// Mitsubishi GX Works2 project: fx1nc_test_in_out   PLC: FX1N/FX1NC

PROGRAM MAIN
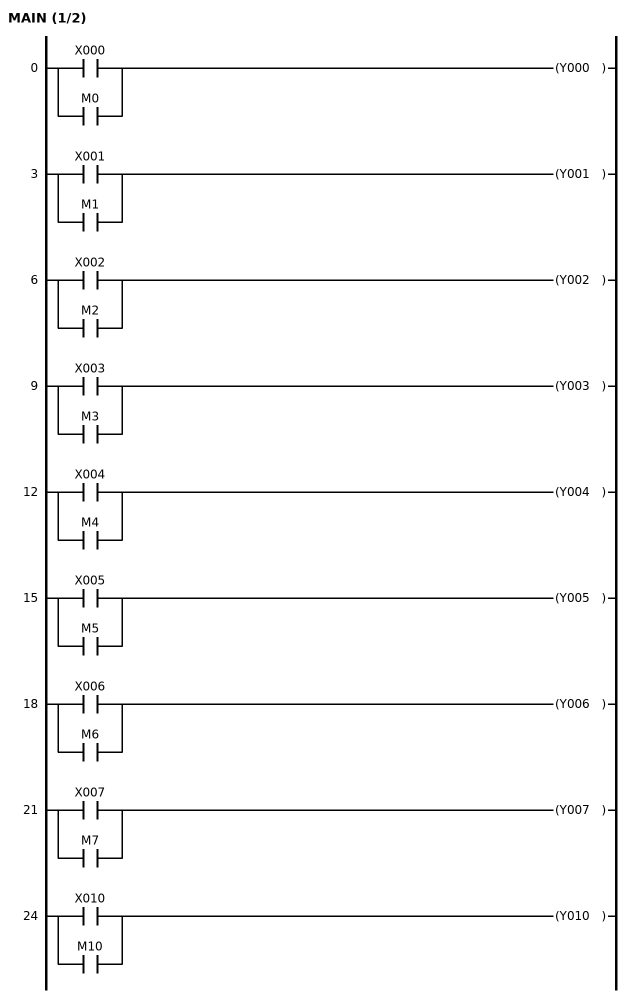
0     LD      X000
      OR      M0
      OUT     Y000
3     LD      X001
      OR      M1
      OUT     Y001
6     LD      X002
      OR      M2
      OUT     Y002
9     LD      X003
      OR      M3
      OUT     Y003
12    LD      X004
      OR      M4
      OUT     Y004
15    LD      X005
      OR      M5
      OUT     Y005
18    LD      X006
      OR      M6
      OUT     Y006
21    LD      X007
      OR      M7
      OUT     Y007
24    LD      X010
      OR      M10
      OUT     Y010
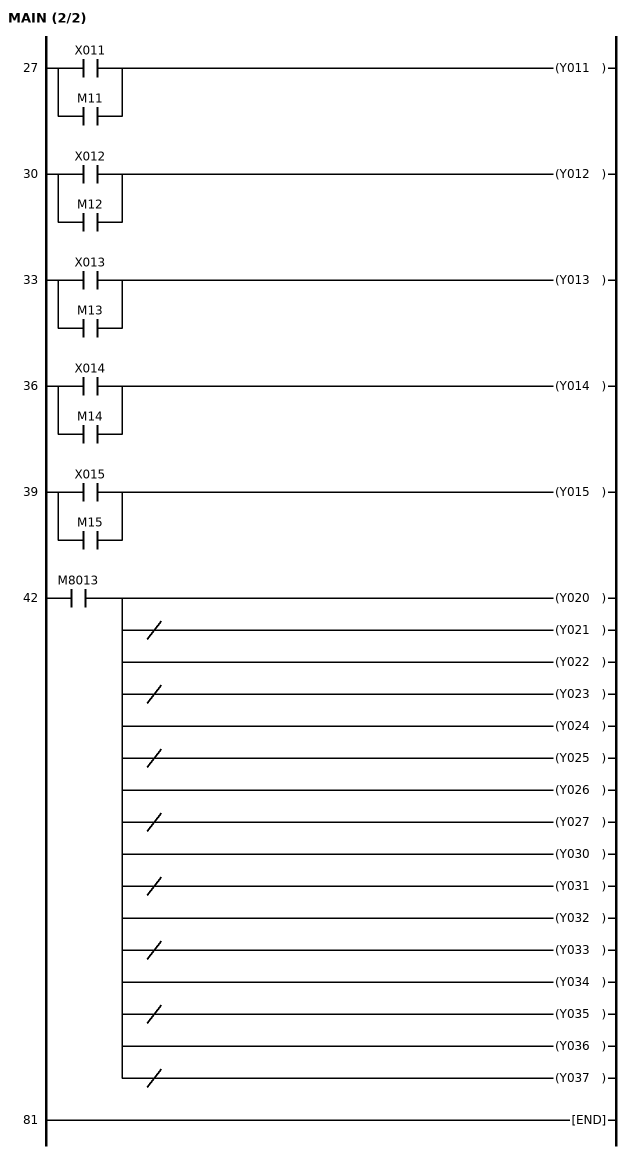
27    LD      X011
      OR      M11
      OUT     Y011
30    LD      X012
      OR      M12
      OUT     Y012
33    LD      X013
      OR      M13
      OUT     Y013
36    LD      X014
      OR      M14
      OUT     Y014
39    LD      X015
      OR      M15
      OUT     Y015
42    LD      M8013
      OUT     Y020
      MPS
      INV
      OUT     Y021
      MPP
      OUT     Y022
      MPS
      INV
      OUT     Y023
      MPP
      OUT     Y024
      MPS
      INV
      OUT     Y025
      MPP
      OUT     Y026
      MPS
      INV
      OUT     Y027
      MPP
      OUT     Y030
      MPS
      INV
      OUT     Y031
      MPP
      OUT     Y032
      MPS
      INV
      OUT     Y033
      MPP
      OUT     Y034
      MPS
      INV
      OUT     Y035
      MPP
      OUT     Y036
      INV
      OUT     Y037
81    END
END_PROGRAM
